(* PLC project TwinForgeCodesysSysModuleBinding, TwinForge TwinForge 0.1.0 *)
(* stored: creationDateTime 2026-07-28T11:19:23.794590+00:00 *)

PROGRAM PLC_PRG
  VAR
    fbModuleBinding : TF_Codesys_ENIP_ModuleBinding;
    xInp_Connected : BOOL;
    xInp_Enabled : BOOL;
    xInp_Faulted : BOOL;
    xInp_DiagnosticAvailable : BOOL;
    xInp_CanReconfigure : BOOL;
    xInp_ReconfigureBusy : BOOL;
    xInp_ReconfigureDone : BOOL;
    xInp_ReconfigureFailed : BOOL;
    xInp_Inhibit : BOOL;
    xInp_Uninhibit : BOOL;
    xOut_Connected : BOOL;
    xOut_Enabled : BOOL;
    xOut_Faulted : BOOL;
    xOut_DiagnosticAvailable : BOOL;
    xOut_RequestReconfigure : BOOL;
    xOut_RequestedEnable : BOOL;
    xOut_ReconfigureBlocked : BOOL;
    xOut_ReconfigureBusy : BOOL;
    xOut_ReconfigureDone : BOOL;
    xOut_ReconfigureFailed : BOOL;
  END_VAR

                  fbModuleBinding(
    Inp_Connected := xInp_Connected,
    Inp_Enabled := xInp_Enabled,
    Inp_Faulted := xInp_Faulted,
    Inp_DiagnosticAvailable := xInp_DiagnosticAvailable,
    Inp_CanReconfigure := xInp_CanReconfigure,
    Inp_ReconfigureBusy := xInp_ReconfigureBusy,
    Inp_ReconfigureDone := xInp_ReconfigureDone,
    Inp_ReconfigureFailed := xInp_ReconfigureFailed,
    Inp_Inhibit := xInp_Inhibit,
    Inp_Uninhibit := xInp_Uninhibit,
    Out_Connected => xOut_Connected,
    Out_Enabled => xOut_Enabled,
    Out_Faulted => xOut_Faulted,
    Out_DiagnosticAvailable => xOut_DiagnosticAvailable,
    Out_RequestReconfigure => xOut_RequestReconfigure,
    Out_RequestedEnable => xOut_RequestedEnable,
    Out_ReconfigureBlocked => xOut_ReconfigureBlocked,
    Out_ReconfigureBusy => xOut_ReconfigureBusy,
    Out_ReconfigureDone => xOut_ReconfigureDone,
    Out_ReconfigureFailed => xOut_ReconfigureFailed
);
                
END_PROGRAM

FUNCTION_BLOCK TF_Codesys_ENIP_ModuleBinding
  VAR_INPUT
    Inp_Connected : BOOL;
    Inp_Enabled : BOOL;
    Inp_Faulted : BOOL;
    Inp_DiagnosticAvailable : BOOL;
    Inp_CanReconfigure : BOOL;
    Inp_ReconfigureBusy : BOOL;
    Inp_ReconfigureDone : BOOL;
    Inp_ReconfigureFailed : BOOL;
    Inp_Inhibit : BOOL;
    Inp_Uninhibit : BOOL;
  END_VAR
  VAR_OUTPUT
    Out_Connected : BOOL;
    Out_Enabled : BOOL;
    Out_Faulted : BOOL;
    Out_DiagnosticAvailable : BOOL;
    Out_RequestReconfigure : BOOL;
    Out_RequestedEnable : BOOL;
    Out_ReconfigureBlocked : BOOL;
    Out_ReconfigureBusy : BOOL;
    Out_ReconfigureDone : BOOL;
    Out_ReconfigureFailed : BOOL;
  END_VAR
  VAR
    CommandLatch : BOOL;
  END_VAR

                  Out_Connected := Inp_Connected;
Out_Enabled := Inp_Enabled;
Out_Faulted := Inp_Faulted;
Out_DiagnosticAvailable := Inp_DiagnosticAvailable;
Out_ReconfigureBusy := Inp_ReconfigureBusy;
Out_ReconfigureDone := Inp_ReconfigureDone;
Out_ReconfigureFailed := Inp_ReconfigureFailed;
Out_RequestReconfigure := FALSE;
IF ((Inp_Inhibit OR Inp_Uninhibit) AND NOT (CommandLatch)) THEN
    IF (Inp_CanReconfigure AND NOT (Inp_ReconfigureBusy)) THEN
        Out_RequestedEnable := NOT (Inp_Inhibit);
        Out_RequestReconfigure := TRUE;
        Out_ReconfigureBlocked := FALSE;
    ELSE
        Out_ReconfigureBlocked := TRUE;
    END_IF;
END_IF;
IF Inp_ReconfigureDone THEN
    Out_ReconfigureBlocked := FALSE;
END_IF;
CommandLatch := (Inp_Inhibit OR Inp_Uninhibit);
                
END_FUNCTION_BLOCK

CONFIGURATION Application
  RESOURCE Application ON PLC
    TASK MainTask(INTERVAL := T#20ms, PRIORITY := 1);
    PROGRAM PLC_PRG WITH MainTask : PLC_PRG;
  END_RESOURCE
END_CONFIGURATION
